Fanuc KAREL source: APPROACH.kl

PROGRAM T
%NOLOCKGROUP
VAR
 v0 : POSITION
 res : VECTOR
BEGIN
 res = APPROACH(v0)
END T
